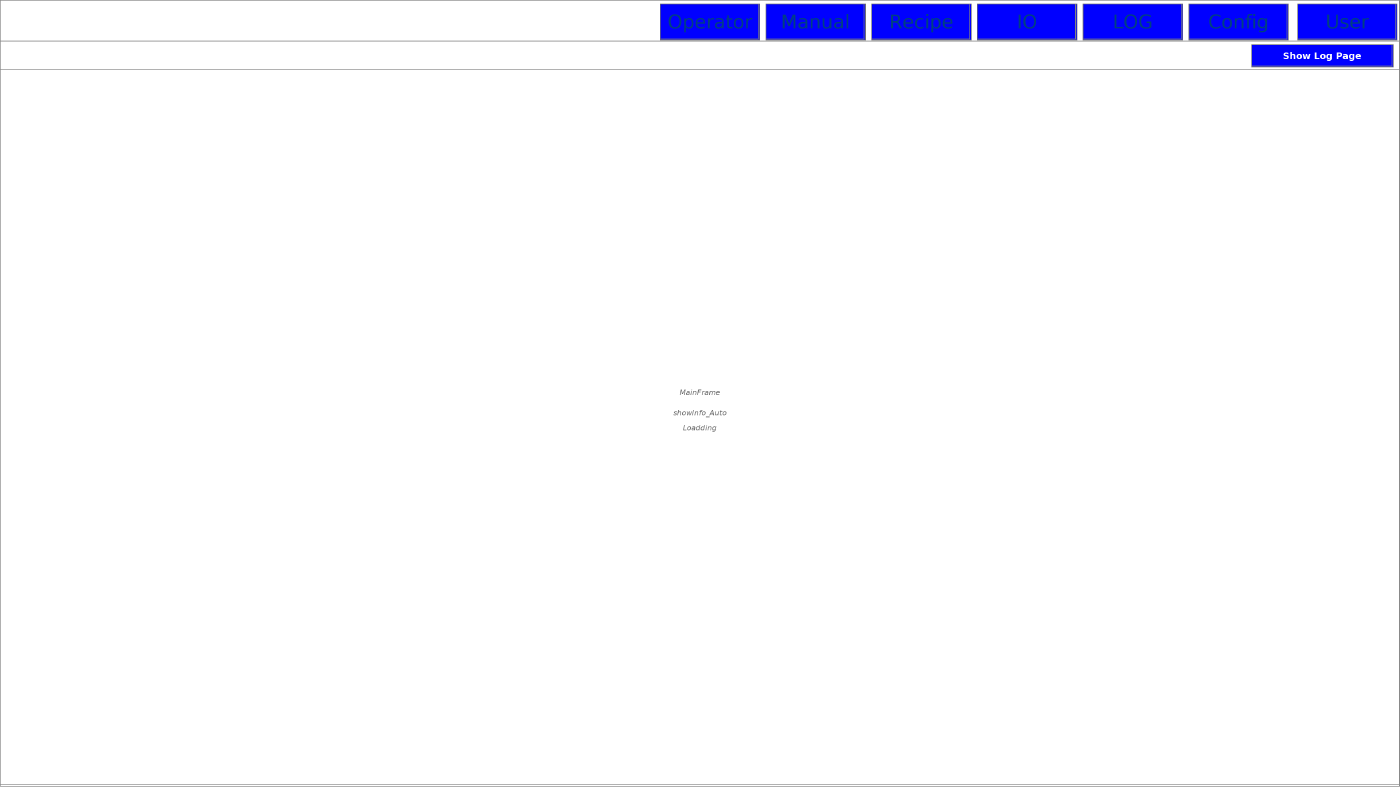
VISUALIZATION Main  // 1920x1080, background image ImagePool1.background
    Frame (0,0 1920x1077)
        shows MainFrame(userData := MainFramDUT)
    Frame (0,95 1920x984)
        shows Loadding()
        shows Manual()
        shows Config()
        shows IO()
        shows LogInf()
        shows Recipe()
        shows Operator()
    Button (1050,5 137x50), "Manual"
        OnMouseClick: execute {
            //MAIN.changePage(1);
        }
        OnMouseClick: FrameSelectionChange Selection=SelectedFrame=81912e38-ebf1-4b8c-bf44-e4a6c92ae24e, Selection=1, GlobSel=AssignType=Directly, SelType=Locally
    Button (1195,5 137x50), "Recipe"
        OnMouseClick: execute {
            //MAIN.changePage(1);
        }
        OnMouseClick: FrameSelectionChange Selection=SelectedFrame=81912e38-ebf1-4b8c-bf44-e4a6c92ae24e, Selection=5, GlobSel=AssignType=Directly, SelType=Locally
    Button (1485,5 137x50), "LOG"
        OnMouseClick: execute {
            //MAIN.changePage(1);
        }
        OnMouseClick: FrameSelectionChange Selection=SelectedFrame=81912e38-ebf1-4b8c-bf44-e4a6c92ae24e, Selection=4, GlobSel=AssignType=Directly, SelType=Locally
    Button (1630,5 137x50), "Config"
        OnMouseClick: execute {
            //MAIN.changePage(1);
        }
        OnMouseClick: FrameSelectionChange Selection=SelectedFrame=81912e38-ebf1-4b8c-bf44-e4a6c92ae24e, Selection=2, GlobSel=AssignType=Directly, SelType=Locally
    Button (1340,5 137x50), "IO"
        OnMouseClick: execute {
            //MAIN.changePage(1);
        }
        OnMouseClick: FrameSelectionChange Selection=SelectedFrame=81912e38-ebf1-4b8c-bf44-e4a6c92ae24e, Selection=3, GlobSel=AssignType=Directly, SelType=Locally
    Button (1779,5 137x50), "User"
        OnMouseClick: execute {
            //MAIN.changePage(1);
        }
        OnMouseClick: FrameSelectionChange Selection=SelectedFrame=81912e38-ebf1-4b8c-bf44-e4a6c92ae24e, GlobSel=AssignType=Directly, SelType=Locally
    Button (905,5 137x50), "Operator"
        OnMouseClick: execute {
            //MAIN.changePage(1);
        }
        OnMouseClick: FrameSelectionChange Selection=SelectedFrame=81912e38-ebf1-4b8c-bf44-e4a6c92ae24e, Selection=6, GlobSel=AssignType=Directly, SelType=Locally
    Frame (0,56 1920x1021), invisible if: (Not gSPOUBusy AND Not gShowPOURunLog) OR ( gSPOUBusy AND Not gShowPOURunLog)
        shows showInfo_Auto(userData := gRunningLog.HMIData)
    Button (1716,61 195x31), "Show Log Page", invisible if: gShowPOURunLog or Not gSPOUBusy
        OnMouseClick: execute { gShowPOURunLog:=NOT gShowPOURunLog; }
END_VISUALIZATION

(* stored: Version 1.1.0.1, ProductVersion 3.1.4024.12
   Visu Main: Id {e8a78d51-3477-4e72-8d40-81ec7501595f} *)
